KUKA KRL data list: msg_wait.dat

&ACCESS RVO11
&REL 17
&COMMENT WARTEN AUF PROZESSSIGNAL
DEFDAT MSG_WAIT
DECL I_MESSAGETYP I_MESSAGE[100]

ENDDAT
